FUNCTION_BLOCK FB_NC_Error

VAR_INPUT
	En				: BOOL;
	nNC_ErrorID	: UDINT;
	nNC_AxisID		: UDINT;
	ErrorSystem		: POINTER TO ST_ErrorSystem;
END_VAR

VAR_OUTPUT
	EnO			: BOOL;
	bError		: BOOL;
END_VAR

VAR
	NCError				: FB_GenericError;
END_VAR



IF En THEN
	EnO	:= En;
	
	IF nNC_ErrorID <> 0 THEN
		NCError.sErrorMessage := 'Axis ';
		NCError.sErrorMessage := CONCAT (NCError.sErrorMessage, UDINT_TO_STRING(nNC_AxisID));
		NCError.sErrorMessage := CONCAT (NCError.sErrorMessage, ' is in error state. NC error ID (Decimal): ');
		NCError.sErrorMessage := CONCAT (NCError.sErrorMessage, UDINT_TO_STRING(nNC_ErrorID));
		NCError.ErrorPriority := 6;
		NCError.bError := TRUE;
	ELSE
		NCError.sErrorMessage := '';
		NCError.bError := FALSE;
		NCError.ErrorPriority := 0;
	END_IF

END_IF

NCError (
	En		:= TRUE,
	bError	:= ,
	sErrorMessage		:= ,
	ErrorPriority		:= ,
	iTerminal_ID		:= ,
	pErrorSystem		:= ErrorSystem,
	EnO		=> ,
);

END_FUNCTION_BLOCK

(* stored: Version 1.1.0.1, ProductVersion 3.1.4022.17
   POU FB_NC_Error: Id {09ed5ba1-d044-4b29-990f-e88331c21ce5}, SpecialFunc None *)
